// TwinCAT 3 PLC project PLC_1
// ProgramVersion: 3.1.4024.0
// libraries:
//   Tc2_ModbusSrv, * (Beckhoff Automation GmbH)
//   Tc2_Standard, * (Beckhoff Automation GmbH)
//   Tc2_System, * (Beckhoff Automation GmbH)
//   Tc3_Module, * (Beckhoff Automation GmbH)
// project tree:
//   GVLs/ GVL.TcGVL
//   / PlcTask.TcTTO
//   POUs/ ButtonController.TcPOU, ConveyorController.TcPOU, EmitterController.TcPOU, MAIN.TcPOU
// real-time tasks:
//   TASK PlcTask: cycle T#10ms, priority 20, ADS port 350

CONFIGURATION PLC_1
    RESOURCE PLC ON TwinCAT3
        TASK PlcTask(INTERVAL := T#10ms, PRIORITY := 20);
        PROGRAM MAIN WITH PlcTask : MAIN;
    END_RESOURCE
END_CONFIGURATION

// ---- GVLs/GVL.TcGVL
{attribute 'qualified_only'}
VAR_GLOBAL
	mb_Input_Coils : ARRAY [0..6] OF BOOL;
	mb_Output_Coils : ARRAY [0..7] OF BOOL;
	isStopON: BOOL;
	isEmgStopON: BOOL;
	isSystemON: BOOL;
	isResetON: BOOL;
	wasEmgBtnPressed: BOOL;
	BlinkBit : BOOL;
END_VAR

// ---- POUs/MAIN.TcPOU
PROGRAM MAIN
VAR
	Start: BOOL;
	Reset: BOOL;
	Stop: BOOL;
	
	StartLight: BOOL;
	ResetLight: BOOL;
	StopLight: BOOL;
	
	AtBufferEntry : BOOL;
	AtBufferExit : BOOL;
	AtExit : BOOL;
	
	Emitter : BOOL;
	EntryConveyor: BOOL;
	ExitConveyor: BOOL;
	EmergencyStop: BOOL;
	
	isStopON: BOOL;
	isEmgStopON: BOOL;
	isSystemON: BOOL;
	isResetON: BOOL;
	wasEmgBtnPressed: BOOL;
	
	ButtonController : ButtonController;
	EmitterController : EmitterController;
	ConveyorController : ConveyorController;
END_VAR

// I/O Assignments
GVL.mb_Input_Coils[1] := StartLight;
GVL.mb_Input_Coils[2] := ResetLight;
GVL.mb_Input_Coils[3] := StopLight;
GVL.mb_Input_Coils[4] := EntryConveyor;
GVL.mb_Input_Coils[5] := ExitConveyor;
GVL.mb_Input_Coils[6] := Emitter;

AtBufferEntry := GVL.mb_Output_Coils[0];
AtBufferExit := GVL.mb_Output_Coils[1];
AtExit := GVL.mb_Output_Coils[2];
Start := gvl.mb_Output_Coils[3];
Reset := gvl.mb_Output_Coils[4];
Stop := gvl.mb_Output_Coils[5];
EmergencyStop := gvl.mb_Output_Coils[7];
// -------------
//Button Control
ButtonController(StartButton := Start, ResetButton := Reset, StopButton := Stop, 
EmgStopButton := EmergencyStop, StartLight => StartLight, ResetLight => ResetLight, StopLight => StopLight);
// -------------
// Emitter Control
EmitterController(AtBufferEntry := AtBufferEntry, Emitter => Emitter);
// -------------
// Conveyor control
ConveyorController(AtBufferEntry := AtBufferEntry, AtBufferExit := AtBufferExit, AtExit := AtExit, EntryConveyor => EntryConveyor, ExitConveyor => ExitConveyor);
// -------------

END_PROGRAM

// ---- POUs/ButtonController.TcPOU
FUNCTION_BLOCK ButtonController
VAR_INPUT
	StartButton: BOOL;
	ResetButton: BOOL;
	StopButton: BOOL;
	EmgStopButton: BOOL;
END_VAR
VAR_OUTPUT
	StartLight: BOOL;
	ResetLight: BOOL;
	StopLight: BOOL;
END_VAR
VAR
	tBlink: TON;
END_VAR

// Blinking logic
tBlink(IN := NOT tBlink.Q, PT := T#1000MS);
GVL.BlinkBit := tBlink.ET > T#500MS;
// -------------
// Memory Bit For SystemON (when true the system is ready to run)
IF GVL.isStopON THEN
	IF NOT GVL.isEmgStopON AND StartButton THEN
		GVL.isSystemON := TRUE;
	END_IF;
END_IF;
IF GVL.isResetON THEN
	IF NOT GVL.isEmgStopON AND StartButton AND NOT GVL.isStopON THEN
		GVL.isSystemON := TRUE;
	END_IF;
END_IF;
IF GVL.isEmgStopON OR NOT StopButton THEN
	GVL.isSystemON := FALSE;
END_IF;
// -------------
// Memory bit for IsEmgStopON - Set/Reset
IF NOT EmgStopButton THEN
	GVL.isEmgStopON := TRUE;
END_IF;
IF EmgStopButton THEN
	GVL.isEmgStopON := FALSE;
END_IF;
// -------------
// Memory bit for IsResetON - Set/Reset
IF ResetButton AND NOT GVL.isEmgStopON AND NOT GVL.isStopON THEN
	GVL.isResetON := TRUE;
END_IF;
IF StartButton THEN
	GVL.isResetON := FALSE;
END_IF;
// -------------
// Memory bit for IsStopON - Set/Reset
IF NOT StopButton AND NOT GVL.isEmgStopON THEN
	GVL.isStopON := TRUE;
END_IF;
IF GVL.isSystemON OR GVL.wasEmgBtnPressed THEN
	GVL.isStopON := FALSE;
END_IF;
// -------------
// Memory bit for wasEmgBtnPressed - Set/Reset
IF NOT EmgStopButton THEN
	GVL.wasEmgBtnPressed := TRUE;
	GVL.isResetON := FALSE;
END_IF;
IF GVL.isSystemON THEN
	GVL.wasEmgBtnPressed := FALSE;
END_IF;
// ------------- OUTPUTS --------------
StartLight := GVL.isSystemON OR ((GVL.isResetON OR (NOT GVL.isResetON AND GVL.isStopON)) AND NOT GVL.isEmgStopON AND NOT GVL.isSystemON AND GVL.BlinkBit);
ResetLight := (GVL.isResetON OR (NOT GVL.isResetON AND GVL.BlinkBit)) AND NOT GVL.isEmgStopON AND NOT GVL.isStopON AND NOT GVL.isSystemON;
StopLight := (GVL.isEmgStopON OR GVL.isStopON) AND NOT GVL.isSystemON;

END_FUNCTION_BLOCK

// ---- POUs/EmitterController.TcPOU
FUNCTION_BLOCK EmitterController
VAR_INPUT
	AtBufferEntry : BOOL;
END_VAR
VAR_OUTPUT
	Emitter : BOOL;
END_VAR
VAR
	TimerTON1 : TON;
	TimerTOF1 : TOF; 
END_VAR

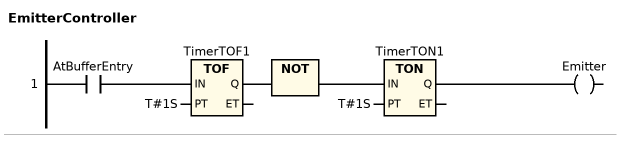
// NETWORK 1
TimerTOF1(IN := AtBufferEntry, PT := T#1S); // TOF
TimerTON1(IN := NOT TimerTOF1.Q, PT := T#1S); // TON
Emitter := TimerTON1.Q;

END_FUNCTION_BLOCK

// ---- POUs/ConveyorController.TcPOU
FUNCTION_BLOCK ConveyorController
VAR_INPUT
	AtBufferEntry : BOOL;
	AtBufferExit : BOOL;
	AtExit : BOOL;
END_VAR
VAR_OUTPUT
	EntryConveyor: BOOL;
	ExitConveyor: BOOL;
END_VAR
VAR
	state: INT;
	TimerTP : TP;
	TimerTOF : TOF;
END_VAR

IF GVL.isSystemON THEN
	CASE state OF
		0: // Box collection stage
			EntryConveyor := TRUE;
			TimerTP(IN := NOT AtBufferExit, PT := T#1200MS, Q => ExitConveyor);
			IF NOT AtExit THEN
				state := 1;
			END_IF;
		1: // Box removal stage
			EntryConveyor := FALSE;
			TimerTOF(IN := NOT AtExit, PT := T#1S, Q => ExitConveyor);
			IF NOT TimerTOF.Q THEN
				state := 0;
			END_IF;
	ELSE
		state := 0;
	END_CASE;
ELSE
	EntryConveyor := FALSE;
	ExitConveyor := FALSE;
	state := 0;
END_IF;

END_FUNCTION_BLOCK
